TYPE DeviceDataEval :
STRUCT
	
	OEM: STRING(50);
	OMEModelName: STRING(50);
	OEMModelCode: STRING(50);
	Model: STRING(50);
	Color: STRING(50);
	OSName: STRING(50);
	OSVersion: STRING(50);
	Profile: STRING(50);
	Carrier: STRING(50);
	IMEI: STRING(30);

END_STRUCT
END_TYPE

(* stored: Version 1.1.0.1, ProductVersion 3.1.4024.6
   DUT DeviceDataEval: Id {bb67c2ec-0ff1-4fca-93d2-caf6e3bed4ea} *)
